PROGRAM MAIN
VAR
END_VAR

PRG_DIAGNOSTIC();
PRG_GATT();

END_PROGRAM

(* stored: Version 1.1.0.1, ProductVersion 3.1.4022.12
   POU MAIN: Id {cd40cec1-86ba-43f9-ae6c-9ca742d8ae87}, SpecialFunc None *)
